// SIMATIC S7-200 project (STEP 7-Micro/WIN), CPU 224 UN REL 02.02

SYMBOL_TABLE USER1
Start            I0.0
S1               I0.3
S2               I0.2
Red              Q0.6
Green            Q0.1
Heater           Q0.7
Pump1            Q0.4
Pump2            Q0.3
mini_pump        Q1.1
D1               I0.6
D2               I0.7
D3               I0.4
Conveyer         Q1.0
END_SYMBOL_TABLE

ORGANIZATION_BLOCK MAIN:OB1
TITLE=PROGRAM COMMENTS
BEGIN
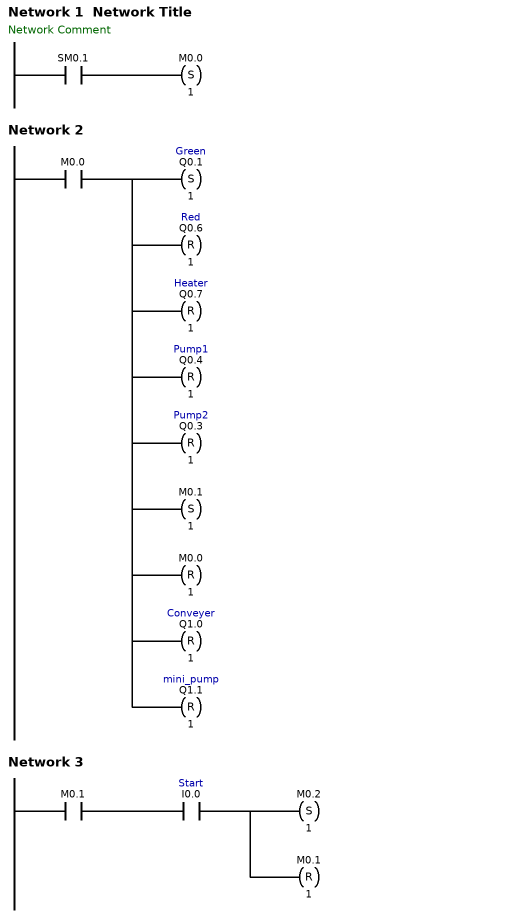
Network 1 // Network Title
// Network Comment
LD     SM0.1
S      M0.0, 1
Network 2
LD     M0.0
S      Green:Q0.1, 1
R      Red:Q0.6, 1
R      Heater:Q0.7, 1
R      Pump1:Q0.4, 1
R      Pump2:Q0.3, 1
S      M0.1, 1
R      M0.0, 1
R      Conveyer:Q1.0, 1
R      mini_pump:Q1.1, 1
Network 3
LD     M0.1
A      Start:I0.0
S      M0.2, 1
R      M0.1, 1
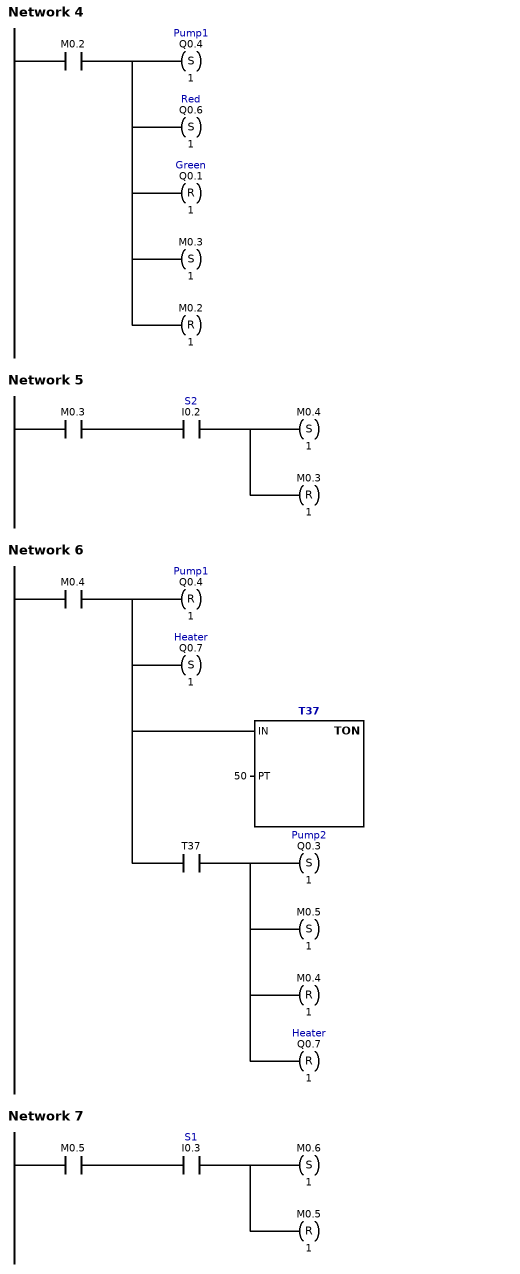
Network 4
LD     M0.2
S      Pump1:Q0.4, 1
S      Red:Q0.6, 1
R      Green:Q0.1, 1
S      M0.3, 1
R      M0.2, 1
Network 5
LD     M0.3
A      S2:I0.2
S      M0.4, 1
R      M0.3, 1
Network 6
LD     M0.4
R      Pump1:Q0.4, 1
S      Heater:Q0.7, 1
TON    T37, 50
A      T37
S      Pump2:Q0.3, 1
S      M0.5, 1
R      M0.4, 1
R      Heater:Q0.7, 1
Network 7
LD     M0.5
A      S1:I0.3
S      M0.6, 1
R      M0.5, 1
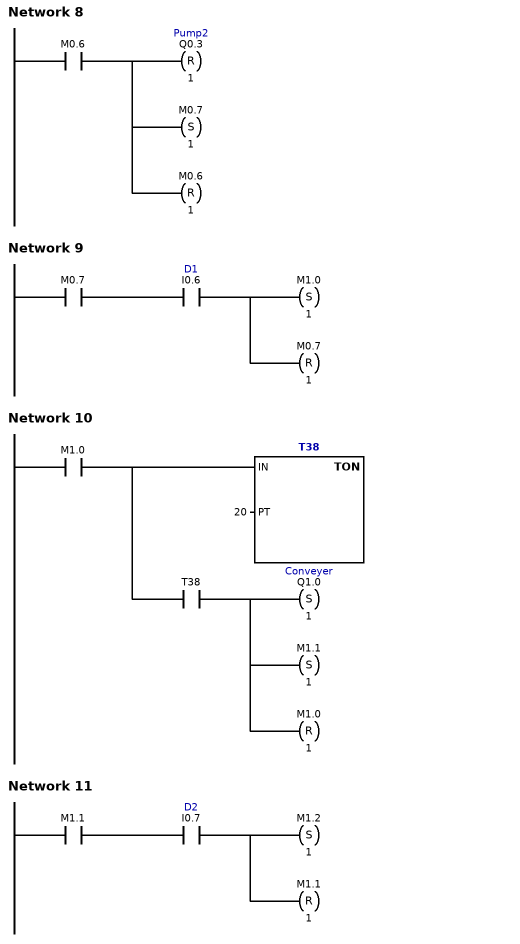
Network 8
LD     M0.6
R      Pump2:Q0.3, 1
S      M0.7, 1
R      M0.6, 1
Network 9
LD     M0.7
A      D1:I0.6
S      M1.0, 1
R      M0.7, 1
Network 10
LD     M1.0
TON    T38, 20
A      T38
S      Conveyer:Q1.0, 1
S      M1.1, 1
R      M1.0, 1
Network 11
LD     M1.1
A      D2:I0.7
S      M1.2, 1
R      M1.1, 1
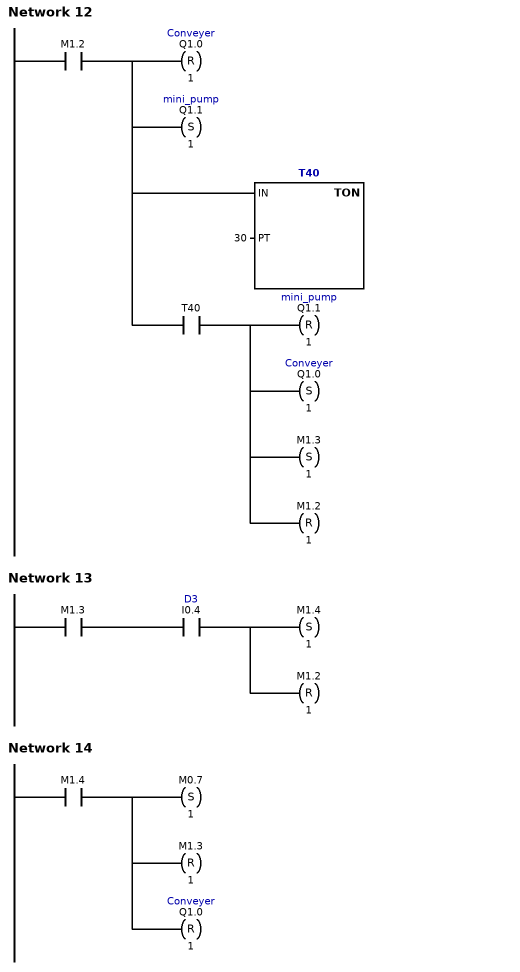
Network 12
LD     M1.2
R      Conveyer:Q1.0, 1
S      mini_pump:Q1.1, 1
TON    T40, 30
A      T40
R      mini_pump:Q1.1, 1
S      Conveyer:Q1.0, 1
S      M1.3, 1
R      M1.2, 1
Network 13
LD     M1.3
A      D3:I0.4
S      M1.4, 1
R      M1.2, 1
Network 14
LD     M1.4
S      M0.7, 1
R      M1.3, 1
R      Conveyer:Q1.0, 1
END_ORGANIZATION_BLOCK
